TYPE
    ST_BoardLengthTestData : STRUCT
        VelocityArray : ARRAY[1..10] OF ST_BoardLengthTest;
    END_STRUCT
END_TYPE

(* stored: Version 1.1.0.1
   DUT ST_BoardLengthTestData: Id {6ebdd11c-2540-4aad-a909-25571dd4d011} *)
